FUNCTION_BLOCK RunCoordinator EXTENDS RunGroupNode
VAR_INPUT
END_VAR
VAR_OUTPUT
END_VAR
VAR
END_VAR

SUPER^();

CASE outputState OF 
	//------------Initialize
	eSpecialStates.GENERIC_GROUP_IDLE:
		//-----------------
		//	IDLE: wait command
		//-----------------
	//------------------------Working
	16#20:
		//------------------
		//	Engineering mode
		//------------------
	16#30:
		//------------------
		//	Daily check mode
		//	1. Bypass some stations
		//  2. Prompt meesage/door interlock
		//  3. Execute SCARA DAILY CHECK
		//------------------
	16#50:
		//---------------------------
		//	Production mode
		//  1. Execute SCARA ASSEMBLE
		//---------------------------
	16#FF:
		//--------------------------------
		//Emergency stop
		// 1. No way out except initialize
		//--------------------------------
END_CASE

END_FUNCTION_BLOCK

(* stored: Version 1.1.0.1, ProductVersion 3.1.4024.0
   POU RunCoordinator: Id {93db79ea-7610-40ae-89e3-5adae225f547}, SpecialFunc None *)
